PROGRAM pouS6Prompts
VAR
	


idbMsgPrompt: FB_CheckMessageBounds;
END_VAR

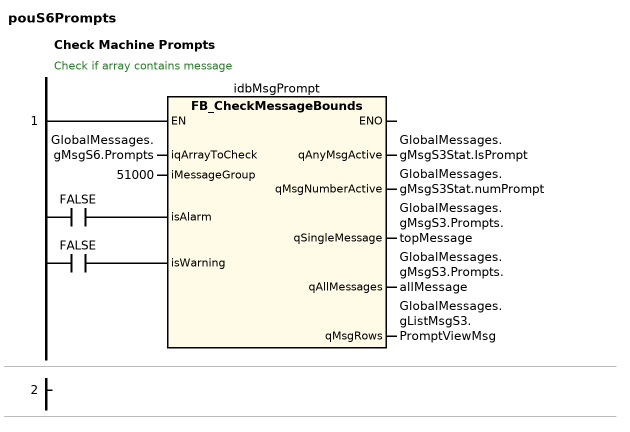
// NETWORK 1: Check Machine Prompts
// Check if array contains message
idbMsgPrompt(
    iqArrayToCheck := GlobalMessages.gMsgS6.Prompts,
    iMessageGroup := 51000,
    isAlarm := FALSE,
    isWarning := FALSE,
    qAnyMsgActive => GlobalMessages.gMsgS3Stat.IsPrompt,
    qMsgNumberActive => GlobalMessages.gMsgS3Stat.numPrompt,
    qSingleMessage => GlobalMessages.gMsgS3.Prompts.topMessage,
    qAllMessages => GlobalMessages.gMsgS3.Prompts.allMessage,
    qMsgRows => GlobalMessages.gListMsgS3.PromptViewMsg); // FB_CheckMessageBounds

// NETWORK 2

END_PROGRAM

(* stored: Version 1.1.0.1, ProductVersion 3.1.4024.12
   POU pouS6Prompts: Id {1b671c62-f677-4124-87af-989471e064aa}, SpecialFunc None *)
